// TwinCAT 3 PLC project Untitled1
// ProgramVersion: 3.1.4024.0
// libraries:
//   Tc2_Standard, * (Beckhoff Automation GmbH)
//   Tc2_System, * (Beckhoff Automation GmbH)
//   Tc3_Module, * (Beckhoff Automation GmbH)
//   VisuDialogs, * (System)
//   VisuSymbols,3.5.10.0,System
// project tree:
//   / GlobalTextList.TcGTLO, PlcTask.TcTTO, Task_Clamp.TcTTO, Task_Saw.TcTTO, Task_SawLengthStop.TcTTO, Task_UserInterface.TcTTO, Visualization Manager.TcVMO (not stored)
//   GVLs/ GVL.TcGVL
//   POUs/ MAIN.TcPOU, POU_MoveToPos.TcPOU, POU_Clamp.TcPOU, POU_Saw.TcPOU, POU_SawLengthStop.TcPOU, POU_UserInterface.TcPOU
//   VISUs/ Visualization.TcVIS, Visualization_1.TcVIS
// real-time tasks:
//   TASK PlcTask: cycle T#10ms, priority 14, ADS port 350
//   TASK Task_Saw: cycle T#10ms, priority 8, ADS port 351
//   TASK Task_Clamp: cycle T#10ms, priority 10, ADS port 352
//   TASK Task_UserInterface: cycle T#10ms, priority 12, ADS port 353
//   TASK Task_SawLengthStop: cycle T#10ms, priority 6, ADS port 354

CONFIGURATION Untitled1
    RESOURCE PLC ON TwinCAT3
        TASK PlcTask(INTERVAL := T#10ms, PRIORITY := 14);
        TASK Task_Clamp(INTERVAL := T#10ms, PRIORITY := 10);
        TASK Task_Saw(INTERVAL := T#10ms, PRIORITY := 8);
        TASK Task_SawLengthStop(INTERVAL := T#10ms, PRIORITY := 6);
        TASK Task_UserInterface(INTERVAL := T#10ms, PRIORITY := 12);
        PROGRAM MAIN WITH PlcTask : MAIN;
        PROGRAM POU_Clamp WITH Task_Clamp : POU_Clamp;
        PROGRAM POU_Saw WITH Task_Saw : POU_Saw;
        PROGRAM POU_SawLengthStop WITH Task_SawLengthStop : POU_SawLengthStop;
        PROGRAM POU_UserInterface WITH Task_UserInterface : POU_UserInterface;
    END_RESOURCE
END_CONFIGURATION

// ---- GVLs/GVL.TcGVL
{attribute 'qualified_only'}
VAR_GLOBAL

	requiredSawingLength : INT;
	startButtonLengthStop: BOOL;
	messageMoveMetalToStop : BOOL;
	startClamp : BOOL;
	sawingProcessDone: BOOL; 
	
	stopPosReached : BOOL;
	metalIsToStop: BOOL;
	
	posReached : BOOL;
	
	clamped: BOOL;
	
	sawingSpeed : INT;
	sawingDone: BOOL;
	bottomPosReached: BOOL;
	
END_VAR

// ---- POUs/MAIN.TcPOU
PROGRAM MAIN
VAR
	counter : INT := 0;
	knop : BOOL :=FALSE;
	lamp :BOOL :=FALSE;
	timer : ton;
	timer1 : ton;
	start_timer: bool;
END_VAR

//counter := counter +1; 

//IF knop THEN
//	lamp :=TRUE;
//ELSE
//	lamp:=FALSE;
//END_IF

END_PROGRAM

// ---- POUs/POU_Clamp.TcPOU
PROGRAM POU_Clamp
VAR
	
	clamping: BOOL;
	clampingDone : bool;
	timer: Ton;
	timerStart : BOOL;
	timerReached: BOOL;
END_VAR

VAR CONSTANT
	clampTime: TIME := T#3S;
END_VAR

clamping := gvl.startClamp;
gvl.clamped := clampingDone;


timer(in:=clamping, pt:=Clamptime);		
IF clamping THEN
	timerstart := TRUE;
	IF timerreached THEN
		timerstart:= FALSE;
	clampingDone := TRUE;
	ELSIF gvl.sawingProcessDone THEN
	clampingDone := FALSE;
	END_IF
END_IF


timer(in:= timerstart, pt:= clamptime, q => timerreached);

END_PROGRAM

// ---- POUs/POU_Saw.TcPOU
PROGRAM POU_Saw
VAR
	sawingSpeed : INT;	
	startSawing: BOOL;
	saw :BOOL;
	actualPos: INT;
	sawingDone: BOOL;
	pou_movetopos1 : pou_movetopos;	
	state : INT;
	bottomposreached: BOOL;
	
	//timers	
	timer1 : ton;

	timer1Start: BOOL;
	time1: TIME;
	timer1Reached :BOOL;	
	
END_VAR

VAR CONSTANT
	bottomPos: INT := 0;
	topPos: INT := 100;
END_VAR

sawingSpeed := gvl.sawingSpeed;
startSawing:= gvl.clamped;
gvl.sawingProcessDone := sawingDone;
GVL.bottomPosReached := bottomposreached;

IF NOT startsawing THEN
	state := 0;
	sawingDone:= FALSE;	
ELSIF state = 0 THEN
	state :=1;
END_IF

CASE state OF
	0:
	;
	1:
		actualpos := 100;
		timer1start:= TRUE;
		time1 := T#2S;
		gvl.metalIsToStop := FALSE;
		IF timer1.q THEN
			timer1start:= FALSE;			
			state:= 2;
			saw := TRUE;
		END_IF
	2:
		Timer1Start := TRUE;
		time1 := T#1S;
		POU_MoveToPos1(actualPos := actualPos, requiredPos := bottomPos, speed := sawingSpeed, newpos => actualpos);
		IF actualpos <= bottompos AND timer1reached THEN
			Timer1Start:=FALSE;
			bottomposreached := TRUE;
			state := 3;
			saw := false;
		END_IF	

	3:
		timer1start:= TRUE;
		time1 := T#2S;
		IF timer1reached THEN
			timer1start:= FALSE;
			state := 4;
		END_IF
	4:
		POU_MoveToPos1(actualPos := actualPos, requiredPos := toppos, speed := sawingSpeed, newpos => actualpos);
	 	IF actualpos >= toppos THEN
			state := 5;
		END_IF
	5:
		Timer1Start:= TRUE;
		time1 := T#2S;
		IF timer1reached THEN
			timer1start:= FALSE;
			sawingDone:= TRUE;
			state := 6;
		END_IF	
	6:
		Timer1Start:= TRUE;
		time1 := T#2S;
		IF timer1reached THEN
			Timer1Start:= FALSE;
			sawingDone:= FALSE;
			state := 0;
		END_IF	
END_CASE

timer1(in:= Timer1Start, pt:= time1, q =>timer1reached);

END_PROGRAM

// ---- POUs/POU_MoveToPos.TcPOU
FUNCTION_BLOCK PUBLIC POU_MoveToPos
VAR_INPUT
	requiredPos: INT;
	actualpos: INT;
	speed: INT;
END_VAR
VAR_OUTPUT	
	newpos : INT;
END_VAR
VAR
	timer1Start: BOOL;
	timer1Reached : BOOL;
	calculatedTime: TIME;

	timer1: ton;
END_VAR


IF timer1.IN = FALSE THEN
	 timer1start:=TRUE;
END_IF
calculatedTime :=INT_TO_TIME(1000/speed);

IF timer1reached THEN
	timer1start:=FALSE;
	IF requiredPos < actualpos THEN
		newpos := actualPos -1;
	ELSIF requiredpos > actualpos THEN
		newpos := actualPos +1; 
	END_IF
ELSE
	newpos := actualpos;
END_IF

timer1(in:= timer1start, pt:= calculatedTime, q=> timer1reached);

END_FUNCTION_BLOCK

// ---- POUs/POU_SawLengthStop.TcPOU
PROGRAM POU_SawLengthStop
VAR
	requiredSawingLength : INT;
	sawingStopPos: int;
	posReached : BOOL;	
	metalAgainstStop: BOOL;
	pou_movetopos1 : pou_movetopos;
END_VAR

VAR CONSTANT
	movingSpeed: INT := 200; // mm/s
END_VAR

requiredSawingLength := gvl.requiredSawingLength;

IF gvl.startButtonLengthStop THEN
	IF requiredSawingLength = sawingStopPos THEN
		posReached := TRUE;
	ELSE
		posReached := FALSE;
		pou_movetopos1(requiredpos := requiredsawinglength, actualpos:= sawingstoppos, speed := movingspeed, newpos => sawingstoppos);
	END_IF
END_IF

IF requiredSawingLength <> sawingStopPos THEN
	posReached := FALSE;
END_IF

IF metalAgainstStop THEN
	gvl.metalIsToStop := TRUE;
ELSE 
	gvl.metalIsToStop := FALSE;
END_IF

gvl.stopposReached := posreached;

END_PROGRAM

// ---- POUs/POU_UserInterface.TcPOU
PROGRAM POU_UserInterface
VAR
	inputSawingLength : INT;
	inputSawingSpeed: INT :=1;
	startButtonLengthStop: BOOL;
	messageMoveMetalToStop : BOOL;
	startClamp : BOOL;
	oilProblem : BOOL;
	sawingDone: BOOL;
	test : INT ;
	timer : ton;
	
	
	signStartClamping: BOOL;
	timerin: BOOL;
	timertime: TIME;
	timerout: BOOL;
END_VAR

gvl.requiredSawingLength := inputSawingLength;
IF startButtonLengthStop THEN
	gvl.startButtonLengthStop := TRUE;
END_IF

IF gvl.stopPosReached and not gvl.metalIsToStop THEN
	gvl.startButtonLengthStop:= FALSE;
	messagemovemetaltostop := TRUE;
ELSE
		messagemovemetaltostop := FALSE;
END_IF

signStartClamping := gvl.metalIsToStop;
gvl.sawingSpeed := inputsawingspeed;

IF  startClamp THEN
	gvl.startClamp := TRUE;
	
END_IF

IF gvl.metalIsToStop THEN
	messagemovemetaltostop := FALSE; 
END_IF

IF gvl.oilProblem THEN
	oilProblem := TRUE;
END_IF

IF gvl.sawingProcessDone THEN
	sawingDone :=TRUE;
	gvl.startClamp := FALSE;
	timerin := TRUE;
	timertime := T#3S;
END_IF

IF timerout THEN
	sawingdone:= FALSE;
	timerin := FALSE;
END_IF

timer(in:= timerin, pt := timertime, q => timerout);

END_PROGRAM

// ---- GlobalTextList.TcGTLO
TEXTLIST GlobalTextList
  882 = '%i length'
  543 = '%i mm'
  515 = '%i speed'
  510 = '%imm'
  454 = 'clamped'
  256 = 'Label'
  353 = 'metal is to stop '
  889 = 'move metal to stop'
  518 = 'push metal to stop'
  621 = 'saw'
  797 = 'saw hight'
  213 = 'sawing done'
  864 = 'sawing length'
  276 = 'sawing speed'
  154 = 'sawing stop pos'
  117 = 'start clamp'
  359 = 'start length stop'
  315 = 'start proces'
END_TEXTLIST

// ---- VISUs/Visualization.TcVIS
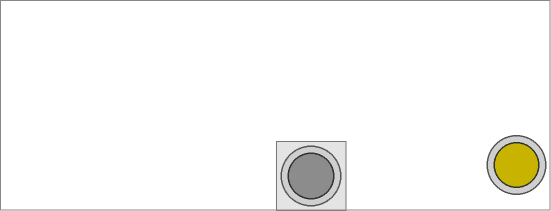
VISUALIZATION Visualization  // 551x211
    PushSwitch (276,141 70x70), variable: GVL.StartButton, behaviour: TOGGLE, style: Switch-PushSwitch-Gray
    Lamp1 (482,130 69x70), variable: GVL.Clamping, style: Lamp-Lamp1-Yellow
END_VISUALIZATION

// ---- VISUs/Visualization_1.TcVIS
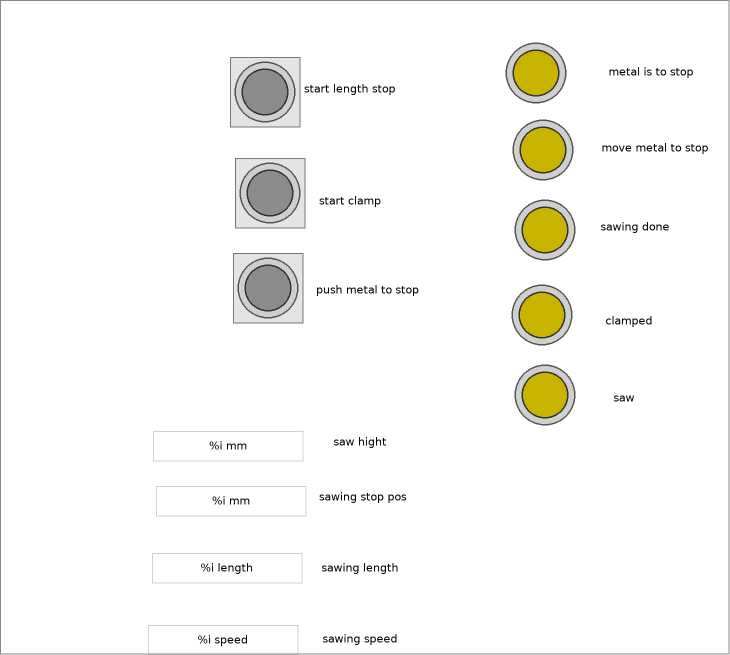
VISUALIZATION Visualization_1  // 730x655
    PushSwitch (230,57 70x70), variable: POU_UserInterface.startButtonLengthStop, behaviour: TOGGLE, style: Switch-PushSwitch-Gray
    Lamp1 (508,115 70x70), variable: POU_UserInterface.messageMoveMetalToStop, style: Lamp-Lamp1-Yellow
    Lamp1 (510,195 70x70), variable: POU_UserInterface.sawingDone, style: Lamp-Lamp1-Yellow
    Textfield (152,553 150x30), "%i length", text variable: POU_UserInterface.inputSawingLength
        OnMouseClick: write the text variable via Default
    Textfield (148,625 150x30), "%i speed", text variable: POU_UserInterface.inputSawingSpeed
        OnMouseClick: write the text variable via Default
    Label (580,133 150x30), "move metal to stop"
    Label (560,212 150x30), "sawing done"
    Label (275,186 150x30), "start clamp"
    Label (288,482 150x30), "sawing stop pos"
    Label (275,74 150x30), "start length stop"
    Label (285,624 150x30), "sawing speed"
    Textfield (156,486 150x30), "%i mm", text variable: POU_SawLengthStop.sawingStopPos
    Label (285,553 150x30), "sawing length"
    PushSwitch (233,253 70x70), variable: POU_SawLengthStop.metalAgainstStop, behaviour: TOGGLE, style: Switch-PushSwitch-Gray
    Label (292,275 151x30), "push metal to stop"
    Lamp1 (501,38 70x70), variable: POU_UserInterface.signStartClamping, style: Lamp-Lamp1-Yellow
    Label (578,57 150x30), "metal is to stop"
    PushSwitch (235,158 70x70), variable: POU_UserInterface.startClamp, behaviour: TOGGLE, style: Switch-PushSwitch-Gray
    Label (285,427 150x30), "saw hight"
    Textfield (153,431 150x30), "%i mm", text variable: POU_Saw.actualPos
    Lamp1 (507,280 70x70), variable: POU_Clamp.clampingDone, style: Lamp-Lamp1-Yellow
    Label (554,306 150x30), "clamped"
    Lamp1 (510,360 70x70), variable: POU_Saw.saw, style: Lamp-Lamp1-Yellow
    Label (549,383 150x30), "saw"
END_VISUALIZATION
